INTERFACE IPredicate EXTENDS IObject

METHOD Check : BOOL
VAR_INPUT
	valueToCompare : __SYSTEM.AnyType; 
END_VAR
END_METHOD

END_INTERFACE

(* stored: Version 1.1.0.1
   Itf IPredicate: Id {2d6a38ba-260b-4d26-a5bc-9bd5e6db19e8}
   Method Check: Id {481953a6-7290-46b0-ac08-ad672ed4bf66} *)
